TYPE ST_EL1008 :
STRUCT
	Input1	: BOOL;
	Input2	: BOOL;
	Input3	: BOOL;
	Input4	: BOOL;
	Input5	: BOOL;
	Input6	: BOOL;
	Input7	: BOOL;
	Input8	: BOOL;
END_STRUCT
END_TYPE

(* stored: Version 1.1.0.1, ProductVersion 3.1.4024.6
   DUT ST_EL1008: Id {6a75c7e6-1478-4c78-a23d-9c06e49e8c48} *)
